ACTION ProcessInit_R1R2:
//*************************************************************************************************************
//
// build configuration for Instances and ProcessInterfaces
//
//*************************************************************************************************************
//*************************************************************************************************************
// - BufferInfeed     : single XtsStation which looks for input trigger from transfersystem, 
//                      transfersystem writes positions of XtsStations to be used at Infeed. 
//                      BufferInfeed is writing ItfProcessCollector[BufferInfeed.ProcessTarget].ActivateStation 
//                        for BufferInfeed target (Infeed / 12 XtsStations).
//                      BufferInfeed sends required amount of movers to WaitPos of XtsStations 
//                        of BufferInfeed target (Infeed / 12 XtsStations).
//-------------------------------------------------------------------------------------------------------------
// whoami
//
// process target (Infeed / 12 XtsStations)
//-------------------------------------------------------------------------------------------------------------
BufferInfeed.ProcessId                    := ProcessCollector[E_INSTANCE.BUFFER_INFEED].ProcessId;
BufferInfeed.ProcessTarget                := ProcessCollector[E_INSTANCE.INFEED].ProcessId;
BufferInfeed.CollectorInterface           := ItfProcessCollector;
BufferInfeed.ProcessLinkedLists           := ItfProcessList;
//-------------------------------------------------------------------------------------------------------------
// configure range of XtsStations for process
//
// see MAIN.StationParameterInit() for positions and dyn constraints
//-------------------------------------------------------------------------------------------------------------
ItfProcessCollector[BufferInfeed.ProcessId].StationFirst  := 53;
ItfProcessCollector[BufferInfeed.ProcessId].StationLast   := 53;

_nStnFrst                                 := ProcessCollector[BufferInfeed.ProcessId].StationFirst;
BufferInfeed.CheckPosition                := 15.0;

//-------------------------------------------------------------------------------------------------------------
//-------------------------------------------------------------------------------------------------------------
//*************************************************************************************************************
//*************************************************************************************************************
// - Infeed         : 12 XtsStations for transfersystem to unload
//                    Infeed is pulling in the movers according to list entry from BufferInfeed
//                    one stop only
//                    must be checked for all mover standstill in PosStop[1] of each XtsStation
//                    must be released by handshake from transfersystem (this is done by a TON for now)
//-------------------------------------------------------------------------------------------------------------
// whoami
//
// process target (BufferOutfeed / 1 XtsStation)
// TODO: 
//    configure infeed target for OUTFEED_CLAMP (12 XtsStations)
//    Infeed.ProcessTarget  := ProcessCollector[E_INSTANCE.OUTFEED_CLAMP].ProcessId;
//-------------------------------------------------------------------------------------------------------------
Infeed.ProcessId                          := ProcessCollector[E_INSTANCE.INFEED].ProcessId;
Infeed.ProcessTarget                      := ProcessCollector[E_INSTANCE.BUFFER_OUTFEED].ProcessId;
Infeed.CollectorInterface                 := ItfProcessCollector;
Infeed.ProcessLinkedLists                 := ItfProcessList;
//-------------------------------------------------------------------------------------------------------------
// configure range of XtsStations for process
//
// see MAIN.StationParameterInit() for positions and dyn constraints
//-------------------------------------------------------------------------------------------------------------
ItfProcessCollector[Infeed.ProcessId].StationFirst        :=  1;
ItfProcessCollector[Infeed.ProcessId].StationLast         := 12;
//-------------------------------------------------------------------------------------------------------------
//-------------------------------------------------------------------------------------------------------------
//*************************************************************************************************************
//*************************************************************************************************************
// - BufferOutfeed  : single XtsStation which distributes movers to specified range 
//                    Infeed sends all movers here 
//                    BufferOutfeed ensures that OutputR2 and OutputR1 have 12 movers each for every job
//                    BufferOutfeed checks if the Queue of this single XtsStation is empty or not
//-------------------------------------------------------------------------------------------------------------
// whoami
//
// process target (Outfeed (OutfeedR2 & OutfeedR1) / 24 XtsStations)
//
//  - optional process target (Outfeed 12 XtsStations)
//-------------------------------------------------------------------------------------------------------------
_nBufferOutfeedTarget[1] := E_INSTANCE.OUTFEED_ROBOT_R1;
_nBufferOutfeedTarget[2] := E_INSTANCE.OUTFEED_ROBOT_R2;

BufferOutfeed.ProcessId              := E_INSTANCE.BUFFER_OUTFEED;
BufferOutfeed.ProcessTarget          := _nBufferOutfeedTarget; 
BufferOutfeed.CollectorInterface     := ItfProcessCollector;
BufferOutfeed.ProcessLinkedLists     := ItfProcessList;
//-------------------------------------------------------------------------------------------------------------
// configure range of XtsStations for process
//
// see MAIN.StationParameterInit() for positions and dyn constraints
//-------------------------------------------------------------------------------------------------------------
ItfProcessCollector[BufferOutfeed.ProcessId].StationFirst  := 25;
ItfProcessCollector[BufferOutfeed.ProcessId].StationLast   := 25;

_nStnFrst                                 := ProcessCollector[BufferOutfeed.ProcessId].StationFirst;
BufferOutfeed.CheckPosition          := 2500.0;
//-------------------------------------------------------------------------------------------------------------
//-------------------------------------------------------------------------------------------------------------
//*************************************************************************************************************
//*************************************************************************************************************
// - Outfeed_R1  : 12 XtsStations for Robot 
//                    All XtsStations must be filled before robot can start 
//                    affter process all movers are sent to Sender process (high speed for the way back)
//                     
//                    
//-------------------------------------------------------------------------------------------------------------
// whoami
//
// process target (SenderFast / 1 XtsStation)
//-------------------------------------------------------------------------------------------------------------
Outfeed_R1.ProcessId                      := E_INSTANCE.OUTFEED_ROBOT_R1;
Outfeed_R1.ProcessTarget                  := ProcessCollector[E_INSTANCE.SENDER_FAST].ProcessId;
Outfeed_R1.CollectorInterface             := ItfProcessCollector;
Outfeed_R1.ProcessLinkedLists             := ItfProcessList;
//-------------------------------------------------------------------------------------------------------------
// configure range of XtsStations for process
//
// see MAIN.StationParameterInit() for positions and dyn constraints
//-------------------------------------------------------------------------------------------------------------
ItfProcessCollector[Outfeed_R1.ProcessId].StationFirst  := 26;
ItfProcessCollector[Outfeed_R1.ProcessId].StationLast   := 37;

_nStnFrst                                 := ProcessCollector[Outfeed_R1.ProcessId].StationFirst;
Outfeed_R1.CheckPosition                  := 6000.0;
//-------------------------------------------------------------------------------------------------------------
//-------------------------------------------------------------------------------------------------------------
//*************************************************************************************************************
//*************************************************************************************************************
// - Outfeed_R2  : 12 XtsStations for Robot 
//                    All XtsStations must be filled before robot can start 
//                    affter process all movers are sent to Sender process (high speed for the way back)
//                     
//                    
//-------------------------------------------------------------------------------------------------------------
// whoami
//
// process target (SenderFast / 1 XtsStation)
//-------------------------------------------------------------------------------------------------------------
Outfeed_R2.ProcessId                      := E_INSTANCE.OUTFEED_ROBOT_R2;
Outfeed_R2.ProcessTarget                  := ProcessCollector[E_INSTANCE.SENDER_FAST].ProcessId;
Outfeed_R2.CollectorInterface             := ItfProcessCollector;
Outfeed_R2.ProcessLinkedLists             := ItfProcessList;
//-------------------------------------------------------------------------------------------------------------
// configure range of XtsStations for process
//
// see MAIN.StationParameterInit() for positions and dyn constraints
//-------------------------------------------------------------------------------------------------------------
ItfProcessCollector[Outfeed_R2.ProcessId].StationFirst  := 38;
ItfProcessCollector[Outfeed_R2.ProcessId].StationLast   := 49;

_nStnFrst                                 := ProcessCollector[Outfeed_R2.ProcessId].StationFirst;
Outfeed_R2.CheckPosition                  := 6000.0;
//-------------------------------------------------------------------------------------------------------------
//-------------------------------------------------------------------------------------------------------------
//*************************************************************************************************************
//*************************************************************************************************************
// - SenderFast  : 1 XtsStation 
//                    movers are handled when entering position area 
//                    movers are accelerated to max speed
//                    movers do not stop here
//                    
//-------------------------------------------------------------------------------------------------------------
// whoami
//
// process target (SenderBufferInfeed / 1 XtsStation)
//-------------------------------------------------------------------------------------------------------------
SenderFast.ProcessId                      := E_INSTANCE.SENDER_FAST;
SenderFast.ProcessTarget                  := ProcessCollector[E_INSTANCE.SENDER_BUFFER_INFEED].ProcessId;
SenderFast.CollectorInterface             := ItfProcessCollector;
SenderFast.ProcessLinkedLists             := ItfProcessList;
//-------------------------------------------------------------------------------------------------------------
// configure range of XtsStations for process
//
// see MAIN.StationParameterInit() for positions and dyn constraints
//-------------------------------------------------------------------------------------------------------------
ItfProcessCollector[SenderFast.ProcessId].StationFirst  := 51;
ItfProcessCollector[SenderFast.ProcessId].StationLast   := 51;

_nStnFrst                                 := ProcessCollector[SenderFast.ProcessId].StationFirst;
SenderFast.CheckPosition                  := GVL_XTS.StationParameter[_nStnFrst].rPosWait - 500.0;
//-------------------------------------------------------------------------------------------------------------
//-------------------------------------------------------------------------------------------------------------
//*************************************************************************************************************
//*************************************************************************************************************
// - SenderBufferInfeed  : 1 XtsStation 
//                    movers are handled when entering position area 
//                    movers are sent to BufferInfeed, so that BufferInfeed has 12 mover ready
//                    movers do stop here, wait until there is room for movers
//                    
//-------------------------------------------------------------------------------------------------------------
// whoami
//
// process target (SenderBufferInfeed / 1 XtsStation)
//-------------------------------------------------------------------------------------------------------------
SenderBufferInfeed.ProcessId              := E_INSTANCE.SENDER_BUFFER_INFEED;
SenderBufferInfeed.ProcessTarget          := ProcessCollector[E_INSTANCE.BUFFER_INFEED].ProcessId;
SenderBufferInfeed.CollectorInterface     := ItfProcessCollector;
SenderBufferInfeed.ProcessLinkedLists     := ItfProcessList;
//-------------------------------------------------------------------------------------------------------------
// configure range of XtsStations for process
//
// see MAIN.StationParameterInit() for positions and dyn constraints
//-------------------------------------------------------------------------------------------------------------
ItfProcessCollector[SenderBufferInfeed.ProcessId].StationFirst  := 52;
ItfProcessCollector[SenderBufferInfeed.ProcessId].StationLast   := 52;

_nStnFrst                                 := ProcessCollector[SenderBufferInfeed.ProcessId].StationFirst;
SenderBufferInfeed.CheckPosition          := GVL_XTS.StationParameter[_nStnFrst].rPosWait - 1250.0;
//-------------------------------------------------------------------------------------------------------------
//-------------------------------------------------------------------------------------------------------------
//*************************************************************************************************************
END_ACTION

END_PROGRAM

// ---- MAIN.TcPOU
//---------------------------------------------------------------------------------------------------------------
//
//  HAUD 2024.03.18
//
//  - XTS_TRANSPORT_LAYER
//  - transport layer members:
//    - CaGroup
//      - access to Group functions
//
//    - Mover
//      - access to MC and CA motion functions
//
//    - Xpu (ProcessingUnit)
//      - access to TcCOM Objects in Environment
//
//    - Transport Control Unit
//      - coordinates members to get XTS in defined states
//
//    - Xts Stations
//      - handshakes with extern control for mover transport
//
//  - global datafields for mrmbers in GVL_XTS namespace
//  - global interface datafields for use in members
//  - structures are assigned by reference for every member
//
//---------------------------------------------------------------------------------------------------------------
// HAUD 2024 05 29
//
//    XTS_TRANSPORT_LAYER project
//    
//    MIT License
//    
//    Copyright (c) 2024 HAUD
//    
//    Permission is hereby granted, free of charge, to any person obtaining a copy
//    of this software and associated documentation files (the "Software"), to deal
//    in the Software without restriction, including without limitation the rights
//    to use, copy, modify, merge, publish, distribute, sublicense, and/or sell
//    copies of the Software, and to permit persons to whom the Software is
//    furnished to do so, subject to the following conditions:
//    
//    The above copyright notice and this permission notice shall be included in all
//    copies or substantial portions of the Software.
//    
//    THE SOFTWARE IS PROVIDED "AS IS", WITHOUT WARRANTY OF ANY KIND, EXPRESS OR
//    IMPLIED, INCLUDING BUT NOT LIMITED TO THE WARRANTIES OF MERCHANTABILITY,
//    FITNESS FOR A PARTICULAR PURPOSE AND NONINFRINGEMENT. IN NO EVENT SHALL THE
//    AUTHORS OR COPYRIGHT HOLDERS BE LIABLE FOR ANY CLAIM, DAMAGES OR OTHER
//    LIABILITY, WHETHER IN AN ACTION OF CONTRACT, TORT OR OTHERWISE, ARISING FROM,
//    OUT OF OR IN CONNECTION WITH THE SOFTWARE OR THE USE OR OTHER DEALINGS IN THE
//    SOFTWARE.
//---------------------------------------------------------------------------------------------------------------
PROGRAM MAIN
VAR
	bInit 				: BOOL;
  eInit         : E_PROGRESS;

  nStation,
	nMover,
  nMoverSelected,
  nStationSelected,
  nStationParameter   : UINT;

  sStationText        : STRING(30);

  eTransportState     : E_XTS_TRANSPORT_STATE;
  eTransportResult    : E_PROGRESS;

  eXpuState           : E_XPU_STATE;
  eXpuResult          : E_PROGRESS;
  eXpuCheck           : E_XPU_CHECK;

  eMoverState         : E_MOVER_STATE;
  eMoverResult        : E_PROGRESS;

  sCaGroupState,
  sTransportState,
  sTransportCheck,
  sTransportResult,
  sXpuState,
  sXpuResult,
  sXpuCheck,
  sXpuOpMode,
  sXpuMoverdetectionMode,
  sXpuMoverAssignement,
  sMoverState,
  sMoverResult,
  sStationState,
  sStationStateMask,
  sStationCtrlMask        : STRING;

  bStationEnable,
  bStationEnter,
  bStationStart,
  bStationDone,
  bStationOut,
  bStationGone            : BOOL;

  tStationSelectedQueue   : ARRAY[1..MAX_LIST_NODES] OF ST_STATION_MOVER_DATA;

  nStn                    : UINT;

  bWriteVariant           : BOOL;
  nParameterVariant       : UINT;
  rAcc                    : REAL := 30000.0;

  eMsgState                   : e_message_state;
  eMsgProgress                : E_PROGRESS;

  eMtrState                   : e_message_state;
  eMtrProgress                : E_PROGRESS;
END_VAR

//############################################################################
// Local time; used for timestamps
//############################################################################
GVL_MSG.fbLocalTime(
                    sLocalTime          => GVL_MSG.sLocalTime, 
                    dtLocalTime         => GVL_MSG.dtLocalTime);
//############################################################################
//############################################################################
// 	example for init sequence
//############################################################################	
IF NOT bInit
THEN
  CASE eInit
  OF
    E_PROGRESS.PROGRESS_INVALID,
    E_PROGRESS.PROGRESS_DONE:         // clear command interface
      eInit                                     := E_PROGRESS.PROGRESS_BUSY;
      GVL_XTS.XpuCtrl.Cmd                       := E_XPU_CTRL.XTS_CMD_NULL;
      GVL_MSG.TransportMessageCtrl.Cmd          := E_MESSAGE_CTRL.MSG_CTRL_NULL;
      GVL_MSG.MetricsMessageCtrl.Cmd            := E_MESSAGE_CTRL.MSG_CTRL_NULL;


      GVL_MSG.MessageLevelXpu                   := E_MessageType.eMessageVerbose; //GVL_MSG.MessageLevel;
      GVL_XTS.CaGroup.MessageLevel              := E_MessageType.eMessageVerbose; //GVL_MSG.MessageLevel;
      GVL_XTS.XtsTransport.MessageLevel         := E_MessageType.eMessageVerbose; //GVL_MSG.MessageLevel;

      FOR nStation := 1 TO MAX_STATION
      DO
        GVL_MSG.MessageLevelStations[nStation]  := E_MessageType.eMessageVerbose; //GVL_MSG.MessageLevel;
      END_FOR
      FOR nMover := 1 TO MAX_MOVER
      DO
        GVL_MSG.MessageLevelMovers[nMover]      := E_MessageType.eMessageVerbose; //GVL_MSG.MessageLevel;
      END_FOR


    E_PROGRESS.PROGRESS_BUSY:         // init Xpu, ProcessingUnit, MotorModules
      eInit                                     := E_PROGRESS.PROGRESS_PREPARE;
      GVL_XTS.XpuCtrl.Cmd                       := E_XPU_CTRL.XTS_CMD_INIT;
      GVL_MSG.TransportMessageCtrl.Cmd          := E_MESSAGE_CTRL.MSG_CTRL_INIT;
      GVL_MSG.MetricsMessageCtrl.Cmd            := E_MESSAGE_CTRL.MSG_CTRL_INIT;


    E_PROGRESS.PROGRESS_PREPARE:      // wait for init to be done
      IF (GVL_XTS.XpuState.State      = E_XPU_STATE.XTS_INIT + E_PROGRESS.PROGRESS_DONE)
      THEN
        eInit                                   := E_PROGRESS.PROGRESS_STARTUP;
        GVL_XTS.XpuCtrl.Cmd                     := E_XPU_CTRL.XTS_IDLE;
      END_IF

    E_PROGRESS.PROGRESS_STARTUP:      // check log file creation and assign mover interfaces
      IF (GVL_MSG.TransportMessageData.FileCreated) AND
         (GVL_MSG.MetricsMessageData.FileCreated)
      THEN
        eInit                                   := E_PROGRESS.PROGRESS_CHECK;
        GVL_MSG.TransportMessageCtrl.Cmd        := E_MESSAGE_CTRL.MSG_CTRL_IDLE;  // one local copy is made, no file is written
        GVL_MSG.MetricsMessageCtrl.Cmd          := E_MESSAGE_CTRL.MSG_CTRL_IDLE;  // one local copy is made, no file is written

        //---------------------------------------------------------------------------------------------------------------------
        // automated file write:
        //---------------------------------------------------------------------------------------------------------------------
        // GVL_MSG.TransportMessageCtrl.Cmd        := E_MESSAGE_CTRL.MSG_CTRL_NULL;  // MessageIndex and ErrorIndex are checked
        // GVL_MSG.MetricsMessageCtrl.Cmd          := E_MESSAGE_CTRL.MSG_CTRL_NULL;  // MessageIndex and ErrorIndex are checked
        //---------------------------------------------------------------------------------------------------------------------
        FOR nMover := 1 TO MAX_MOVER
        DO
          GVL_XTS.MoverItf[nMover]              := GVL_XTS.Mover[nMover];
        END_FOR
      END_IF

    E_PROGRESS.PROGRESS_CHECK:        // assign CaGroup interface
      eInit                                     := E_PROGRESS.PROGRESS_OCCUPIED;
      GVL_XTS.CaGroupItf                        := GVL_XTS.CaGroup;

    E_PROGRESS.PROGRESS_OCCUPIED:     // StartStation for XtsTransportCtrl.Cmd := E_XTS_TRANSPORT_CTRL.CMD_TRANSPORT_START;
      bWriteVariant                             := TRUE;
      eInit                                     := E_PROGRESS.PROGRESS_WORKING;

      // where to start?
      GVL_XTS.XtsTransport.StationStartIndex    := GVL_XTS.StationStartIndex;

      GVL_MSG.MessageLevelXpu                   := GVL_MSG.MessageLevel;
      GVL_XTS.CaGroup.MessageLevel              := GVL_MSG.MessageLevel;
      GVL_XTS.XtsTransport.MessageLevel         := GVL_MSG.MessageLevel;

      FOR nStation := 1 TO MAX_STATION
      DO
        GVL_MSG.MessageLevelStations[nStation]  := GVL_MSG.MessageLevel;
      END_FOR
      FOR nMover := 1 TO MAX_MOVER
      DO
        GVL_MSG.MessageLevelMovers[nMover]      := GVL_MSG.MessageLevel;
      END_FOR

    E_PROGRESS.PROGRESS_WORKING:
      // Start Position parameters
      GVL_XTS.StationStart.rPosWait             :=  20500.0; // this value may differ from the GVL_XTS.StationParameter[StartStationIndex], IF it differs, you MUST have room for positive movement to GVL_XTS.StationParameter[StartStationIndex].rWaitPos
      GVL_XTS.StationStart.rGap                 :=     85.0; // may differ, or just copy from GVL_XTS.StationParameter[StartStationIndex]
      GVL_XTS.StationStart.rVelo                :=   1250.0; // may differ, or just copy from GVL_XTS.StationParameter[StartStationIndex]
      GVL_XTS.StationStart.rAccDec              :=  15000.0; // may differ, or just copy from GVL_XTS.StationParameter[StartStationIndex]
      GVL_XTS.StationStart.rJerk                := 400000.0; // may differ, or just copy from GVL_XTS.StationParameter[StartStationIndex], the movements are more robust if you keep this value in a narrow range, since jumps lead to adjusting movements within the CA Group

      IF (GVL_XTS.XtsTransport.StationStartIndex > 0) AND
         (GVL_XTS.XtsTransport.StationStartIndex < MAX_STATION+1)
      THEN
        GVL_XTS.StationStart.nConfiguredStopCount := GVL_XTS.StationParameter[GVL_XTS.XtsTransport.StationStartIndex].nConfiguredStopCount;
      END_IF

      bInit                                     := TRUE;
      eInit                                     := E_PROGRESS.PROGRESS_DONE;
  END_CASE
END_IF
//############################################################################
//############################################################################
// 	XTS Transport Unit
//############################################################################
//  - main control function block for transport layer
//  - requires access to member controls
//    - Xpu
//    - CaGroup
//    - Mover
//    - Station Control
//    - Station LinkedList Interface
//############################################################################
//
// cyclic call
GVL_XTS.XtsTransport();

// main control
GVL_XTS.XtsTransport.Ctrl               REF= GVL_XTS.XtsTransportCtrl;   // main control
GVL_XTS.XtsTransport.State              REF= GVL_XTS.XtsTransportState;  // main state
                                        
// member controls                      
GVL_XTS.XtsTransport.XpuCtrl            REF= GVL_XTS.XpuCtrl;
GVL_XTS.XtsTransport.XpuState           REF= GVL_XTS.XpuState;
GVL_XTS.XtsTransport.XpuInfo            REF= GVL_XTS.XpuInfo;
                                        
GVL_XTS.XtsTransport.GroupItf           :=   GVL_XTS.CaGroupItf;
GVL_XTS.XtsTransport.GroupInfo          REF= GVL_XTS.CaGroupInfo;
                                        
GVL_XTS.XtsTransport.MoverItf           REF= GVL_XTS.MoverItf;
GVL_XTS.XtsTransport.MoverInfo          REF= GVL_XTS.MoverInfo;
GVL_XTS.XtsTransport.MoverLastPosition  REF= GVL_XTS.LastPosition;
GVL_XTS.XtsTransport.MoverLastGap       REF= GVL_XTS.LastGap;
                                        
GVL_XTS.XtsTransport.StationStart       REF= GVL_XTS.StationStart;      // start position for E_XTS_TRANSPORT_CTRL.CMD_TRANSPORT_START
GVL_XTS.XtsTransport.StationCtrlItf     REF= GVL_XTS.StationCtrlItf;    // station interfaces are required for accessing station methods
GVL_XTS.XtsTransport.StationListsItf    REF= GVL_XTS.StationListItf;    // list interface is required for access to linked list methods
GVL_XTS.XtsTransport.StationControl     REF= GVL_XTS.StationCtrl;
GVL_XTS.XtsTransport.StationState       REF= GVL_XTS.StationState;
//############################################################################



//############################################################################
// 	XTS Stations
//############################################################################	
FOR nStation := 1 TO MAX_STATION
DO
  GVL_XTS.Station[nStation].StationId   := nStation;
  GVL_XTS.Station[nStation].MessageLevel:= GVL_MSG.MessageLevelStations[nStation];

  GVL_XTS.StationListItf[nStation]      := GVL_XTS.StationList[nStation];   // interfaces for list methods
  GVL_XTS.StationCtrlItf[nStation]      := GVL_XTS.Station[nStation];       // interfaces for station methods

  GVL_XTS.Station[nStation].Ctrl        REF= GVL_XTS.StationCtrl;           // station ctrl from extern
  GVL_XTS.Station[nStation].State       REF= GVL_XTS.StationState;          // station state to extern

  GVL_XTS.Station[nStation].ItfStations REF= GVL_XTS.StationListItf;        // give every station all list interfaces for writing mover tickets
  GVL_XTS.Station[nStation].ItfMover    REF= GVL_XTS.MoverItf;              // give every station all mover interfaces for movement in / out of station
  GVL_XTS.Station[nStation].Mover       REF= GVL_XTS.AxisRefMover;          // AXIS_REF to read infos from
  GVL_XTS.Station[nStation].MoverOffset REF= GVL_XTS.PositionOffset;        // static offsets for all stations, all movers, all stop positions


  GVL_XTS.Station[nStation].StationParameter  REF= GVL_XTS.StationParameter;// give every station all station parameters for sending to WaitPos of target station

  // cyclic call
  GVL_XTS.Station[nStation].Cycle();                                        // cycle for handshaking with extern

  // Queue data for each station
  GVL_XTS.StationQueue[nStation]        := GVL_XTS.StationListItf[nStation].Data;
END_FOR
//############################################################################



//############################################################################
// 	XPU environment
//############################################################################	
GVL_XTS.Xpu.XpuInstance                 :=   1;
GVL_XTS.Xpu.MessageLevel                :=   GVL_MSG.MessageLevelXpu;

GVL_XTS.Xpu.Ctrl                        REF= GVL_XTS.XpuCtrl;
GVL_XTS.Xpu.State                       REF= GVL_XTS.XpuState;
GVL_XTS.Xpu.XpuModuleInfoData           REF= GVL_XTS.XpuModules;

GVL_XTS.Xpu.CaGroupOID                  :=   GVL_XTS.CaGroup.GroupInfo.CaGroupOID;

// cyclic call
GVL_XTS.Xpu();
GVL_XTS.XpuInfo                         :=   GVL_XTS.Xpu.XpuInfo;
//############################################################################


//############################################################################	
// 	CA-Group Class
//############################################################################	
// assignment
GVL_XTS.CaGroup.AxisRef                 REF= GVL_XTS.AxisRefMover;
// Interface to Mover methods
GVL_XTS.CaGroup.MoverItf                REF= GVL_XTS.MoverItf; 

GVL_XTS.CaGroup.GroupRef                REF= GVL_XTS.CaGroupRef;

// cyclic call
GVL_XTS.CaGroup.InfoCycle(TRUE); // read group status

// InfoData from group
GVL_XTS.CaGroupInfo                     :=   GVL_XTS.CaGroup.GroupInfo;

// Interface of CaGroup
GVL_XTS.CaGroupItf                      :=   GVL_XTS.CaGroup;
//############################################################################


//############################################################################
// Mover Class	
//############################################################################	
FOR nMover := 1 TO MAX_MOVER
DO
  GVL_XTS.Mover[nMover].MoverId         :=   nMover;
  GVL_XTS.Mover[nMover].RailLength      :=   GVL_XTS.Xpu.RailLength;  // mover needs RailLength, in order to calc absolute position from modulo input
  GVL_XTS.Mover[nMover].MessageLevel    :=   GVL_MSG.MessageLevelMovers[nMover];

  GVL_XTS.Mover[nMover].Ctrl            REF= GVL_XTS.MoverCtrl;       // mover control from extern
  GVL_XTS.Mover[nMover].State           REF= GVL_XTS.MoverState;      // mover state to extern

  GVL_XTS.Mover[nMover].MoveData        REF= GVL_XTS.MoveData;        // dyn constraints for extern to write
  GVL_XTS.Mover[nMover].GearData        REF= GVL_XTS.GearData;        // GearIn/GearInPosCa data fro extern to write

  // assignment	
  GVL_XTS.Mover[nMover].Mover           REF= GVL_XTS.AxisRefMover[nMover];  // axis reference to Mover function block
  GVL_XTS.Mover[nMover].LastGap         REF= GVL_XTS.LastGap[nMover];       // reference to last used gap value datafield
  GVL_XTS.Mover[nMover].LastPosition    REF= GVL_XTS.LastPosition[nMover];  // reference to last position datafield

  GVL_XTS.Mover[nMover].MoverInfo		    REF= GVL_XTS.MoverInfo[nMover];     // refernence to mover info data (ActPos, SetPos, ...)

  GVL_XTS.MoverItf[nMover]              :=   GVL_XTS.Mover[nMover];

  // cyclic call
  GVL_XTS.Mover[nMover].Cycle();  // call AXIS_REF()
  GVL_XTS.Mover[nMover]();        // call Ctrl/State
END_FOR
//############################################################################
//############################################################################
// /logging
//############################################################################
GVL_MSG.TransportMessageData.Ctrl             REF= GVL_MSG.TransportMessageCtrl;
GVL_MSG.TransportMessageData.State            REF= GVL_MSG.TransportMessageState;

GVL_MSG.TransportMessageData.MessageIndex     REF= GVL_MSG.MessageTransportIndex;
GVL_MSG.TransportMessageData.ErrorIndex       REF= GVL_MSG.MessageTransportError;

GVL_MSG.TransportMessageData.DirRoot          :=   ADR(GVL_MSG.LOG_DIR);
GVL_MSG.TransportMessageData.FileRoot         :=   ADR(GVL_MSG.LOG_FILE);

GVL_MSG.TransportMessageData.MsgList          :=   ADR(GVL_MSG.TransportMessages);
GVL_MSG.TransportMessageData.LocalTime        :=   ADR(GVL_MSG.dtLocalTime);

GVL_MSG.TransportMessageData();               

eMsgState                                     := f_GetState   (GVL_MSG.TransportMessageState.State);
eMsgProgress                                  := f_GetProgress(GVL_MSG.TransportMessageState.State);

CASE eMsgState
OF
  E_MESSAGE_STATE.MSG_STATE_NULL:
    CASE eMsgProgress
    OF
      E_PROGRESS.PROGRESS_INVALID,
      E_PROGRESS.PROGRESS_DONE:
        IF (GVL_MSG.MessageTransportIndex > GVL_MSG.MAX_MESSAGE/100) OR
           (GVL_MSG.MessageTransportError > 0)
        THEN
          GVL_MSG.TransportMessageCtrl.Cmd    := E_MESSAGE_CTRL.MSG_CTRL_WRITE;
        END_IF
    END_CASE

  E_MESSAGE_STATE.MSG_STATE_WRITE:
    CASE eMsgProgress
    OF
      E_PROGRESS.PROGRESS_ERROR,
      E_PROGRESS.PROGRESS_DONE:
        GVL_MSG.TransportMessageCtrl.Cmd      := E_MESSAGE_CTRL.MSG_CTRL_NULL;
    END_CASE

ELSE
    CASE eMsgProgress
    OF
      E_PROGRESS.PROGRESS_DONE:
        GVL_MSG.TransportMessageCtrl.Cmd      := E_MESSAGE_CTRL.MSG_CTRL_NULL;
    END_CASE
END_CASE
//############################################################################
// logging/
//############################################################################
//############################################################################
//############################################################################
// /Transport Metrics
//############################################################################
GVL_MSG.MetricsMessageData.Ctrl               REF= GVL_MSG.MetricsMessageCtrl;
GVL_MSG.MetricsMessageData.State              REF= GVL_MSG.MetricsMessageState;

GVL_MSG.MetricsMessageData.MessageIndex       REF= GVL_MSG.MessageMetricsIndex;
GVL_MSG.MetricsMessageData.ErrorIndex         REF= GVL_MSG.MessageMetricsError;

GVL_MSG.MetricsMessageData.DirRoot            :=   ADR(GVL_MSG.LOG_DIR);
GVL_MSG.MetricsMessageData.FileRoot           :=   ADR(GVL_MSG.LOG_FILE_METRIC);

GVL_MSG.MetricsMessageData.MsgList            :=   ADR(GVL_MSG.MetricsMessages);
GVL_MSG.MetricsMessageData.LocalTime          :=   ADR(GVL_MSG.dtLocalTime);

GVL_MSG.MetricsMessageData();

eMtrState                                     := f_GetState   (GVL_MSG.MetricsMessageState.State);
eMtrProgress                                  := f_GetProgress(GVL_MSG.MetricsMessageState.State);

CASE eMtrState
OF
  E_MESSAGE_STATE.MSG_STATE_NULL:
    CASE eMtrProgress
    OF
      E_PROGRESS.PROGRESS_INVALID:
        IF (GVL_MSG.MessageMetricsIndex > 10) OR
           (GVL_MSG.MessageMetricsError > 0)
        THEN
          GVL_MSG.MetricsMessageCtrl.Cmd      := E_MESSAGE_CTRL.MSG_CTRL_WRITE;
        END_IF
    END_CASE

  E_MESSAGE_STATE.MSG_STATE_WRITE:
    CASE eMtrProgress
    OF
      E_PROGRESS.PROGRESS_ERROR,
      E_PROGRESS.PROGRESS_DONE:
        GVL_MSG.MetricsMessageCtrl.Cmd        := E_MESSAGE_CTRL.MSG_CTRL_NULL;
    END_CASE
ELSE
    CASE eMtrProgress
    OF
      E_PROGRESS.PROGRESS_DONE:
        GVL_MSG.MetricsMessageCtrl.Cmd        := E_MESSAGE_CTRL.MSG_CTRL_NULL;
    END_CASE
END_CASE
//############################################################################
// Transport Metrics/
//############################################################################
//############################################################################
//############################################################################
// Visualization data	
//############################################################################	
// get enumerations from XPU for visu:
eTransportState                         := f_GetState   (GVL_XTS.XtsTransportState.State);
eTransportResult                        := f_GetProgress(GVL_XTS.XtsTransportState.State);

eXpuState                               := f_GetState   (GVL_XTS.XpuState.State);
eXpuResult                              := f_GetProgress(GVL_XTS.XpuState.State);

eXpuCheck                               := GVL_XTS.XpuState.Check;

// display xpu state and result in visu
// get strings and info
sCaGroupState                           := TO_STRING(GVL_XTS.CaGroupInfo.CaGroupState);

sTransportState                         := TO_STRING(eTransportState);
sTransportCheck                         := TO_STRING(GVL_XTS.XtsTransportState.Check);
sTransportResult                        := TO_STRING(eTransportResult);

sXpuState                               := TO_STRING(eXpuState);
sXpuResult                              := TO_STRING(eXpuResult);
sXpuCheck                               := TO_STRING(eXpuCheck);

sXpuOpMode                              := GVL_XTS.Xpu.OpModeToString();
sXpuMoverdetectionMode                  := GVL_XTS.Xpu.IdDetectionModeToString();
sXpuMoverAssignement                    := GVL_XTS.Xpu.MoverPositionAssignementToString();

nMoverSelected                          := SEL((nMoverSelected<1), nMoverSelected, 1);
nMoverSelected                          := SEL((nMoverSelected>MAX_MOVER), nMoverSelected, MAX_MOVER);

nStationSelected                        := SEL((nStationSelected<1), nStationSelected, 1);
nStationSelected                        := SEL((nStationSelected>MAX_STATION), nStationSelected, MAX_STATION);

bStationEnable                          := SEL((GVL_XTS.StationCtrl[nStationSelected].eCmd = E_STATION_CTRL.STATION_ENABLE),        FALSE, TRUE);
bStationEnter                           := SEL((GVL_XTS.StationCtrl[nStationSelected].eCmd = E_STATION_CTRL.STATION_MOVER_ENTER),   FALSE, TRUE);
bStationStart                           := SEL((GVL_XTS.StationCtrl[nStationSelected].eCmd = E_STATION_CTRL.STATION_PROCESS_START), FALSE, TRUE);
bStationDone                            := SEL((GVL_XTS.StationCtrl[nStationSelected].eCmd = E_STATION_CTRL.STATION_PROCESS_DONE),  FALSE, TRUE);
bStationOut                             := SEL((GVL_XTS.StationCtrl[nStationSelected].eCmd = E_STATION_CTRL.STATION_MOVER_OUT),     FALSE, TRUE);
bStationGone                            := SEL((GVL_XTS.StationCtrl[nStationSelected].eCmd = E_STATION_CTRL.STATION_MOVER_GONE),    FALSE, TRUE);

eMoverState                             := f_GetState   (GVL_XTS.MoverState[nMoverSelected].State);
eMoverResult                            := f_GetProgress(GVL_XTS.MoverState[nMoverSelected].State);

sMoverState                             := TO_STRING(eMoverState);
sMoverResult                            := TO_STRING(eMoverResult);

sStationState                           := TO_STRING(GVL_XTS.StationState[nStationSelected].eState);
sStationStateMask                       := Tc2_Utilities.BYTE_TO_BINSTR(GVL_XTS.StationState[nStationSelected].nMask, 8);
sStationCtrlMask                        := Tc2_Utilities.BYTE_TO_BINSTR(GVL_XTS.StationCtrl[nStationSelected].nMask, 8);

tStationSelectedQueue                   := GVL_XTS.StationQueue[nStationSelected];

IF bWriteVariant
THEN
  bWriteVariant                         := FALSE;

  CASE nParameterVariant
  OF
    1:
      J_100000_V3000();     // J 100_000 V3000
    2:
      J_100000_V3500();     // J 100_000 V3500
    3:
      J_100000_V4000();     // J 100_000 V4000
    4:
      J_200000_V3000();     // J 200_000 V3000
    5:
      StationParameterInit_4();   // J 400_000
    6:
      StationParameterInit_5();   // J 100_000 PosStop INFEED == 0.0
  ELSE
      StationParameterInit_5();   // J 100_000 PosStop INFEED == 0.0
  END_CASE
END_IF
//############################################################################
//############################################################################

ACTION J_100000_V3000:
//-----------------------------------------------------------------------------
//
//  HAUD 2024.06.12
//
// 
//  - hard coded station parameter
//-----------------------------------------------------------------------------
//-----------------------------------------------------------------------------

FOR nStationParameter := 1 TO MAX_STATION
DO
  GVL_XTS.StationParameter[nStationParameter].rVelo               :=   3000.0;
  GVL_XTS.StationParameter[nStationParameter].rAccDec             := rAcc;
  GVL_XTS.StationParameter[nStationParameter].rJerk               := 100000.0;
END_FOR 

//-----------------------------------------------------------------------------------------------------------------------------------------
//  INFEED
    sStationText  := TO_STRING(E_INSTANCE.INFEED);//'INFEED';
//-----------------------------------------------------------------------------------------------------------------------------------------
nStationParameter := 1;
GVL_XTS.StationParameter[nStationParameter].sText                 := sStationText;
GVL_XTS.StationParameter[nStationParameter].rPosWait              :=    1250.0;  // absolute modulo position

GVL_XTS.StationParameter[nStationParameter].nConfiguredStopCount  :=      1;   // how many stops the mover has to make in this station
GVL_XTS.StationParameter[nStationParameter].rPosStop[1]           :=      0.0 + 176.0; // relative to rPosWait

GVL_XTS.StationParameter[nStationParameter].rReleaseDistance      :=    300.0; // relative to Mover.ActPos
GVL_XTS.StationParameter[nStationParameter].rGap                  :=     76.0;

//-----------------------------------------------------------------------------------------------------------------------------------------
nStationParameter := 2;
GVL_XTS.StationParameter[nStationParameter].sText                 := sStationText;
GVL_XTS.StationParameter[nStationParameter].rPosWait              :=    1250.0; // absolute modulo position

GVL_XTS.StationParameter[nStationParameter].nConfiguredStopCount  :=      1;   // how many stops the mover has to make in this station
GVL_XTS.StationParameter[nStationParameter].rPosStop[1]           :=     76.0 + 176.0; // relative to rPosWait

GVL_XTS.StationParameter[nStationParameter].rReleaseDistance      :=    275.0; // relative to Mover.ActPos
GVL_XTS.StationParameter[nStationParameter].rGap                  :=     76.0;

//-----------------------------------------------------------------------------------------------------------------------------------------
nStationParameter := 3;
GVL_XTS.StationParameter[nStationParameter].sText                 := sStationText;
GVL_XTS.StationParameter[nStationParameter].rPosWait              :=    1250.0; // absolute modulo position

GVL_XTS.StationParameter[nStationParameter].nConfiguredStopCount  :=      1;   // how many stops the mover has to make in this station
GVL_XTS.StationParameter[nStationParameter].rPosStop[1]           :=    152.0 + 176.0; // relative to rPosWait

GVL_XTS.StationParameter[nStationParameter].rReleaseDistance      :=    250.0; // relative to Mover.ActPos
GVL_XTS.StationParameter[nStationParameter].rGap                  :=     76.0;

//-----------------------------------------------------------------------------------------------------------------------------------------
nStationParameter := 4;
GVL_XTS.StationParameter[nStationParameter].sText                 := sStationText;
GVL_XTS.StationParameter[nStationParameter].rPosWait              :=   1250.0;  // absolute modulo position

GVL_XTS.StationParameter[nStationParameter].nConfiguredStopCount  :=      1;   // how many stops the mover has to make in this station
GVL_XTS.StationParameter[nStationParameter].rPosStop[1]           :=    228.0 + 176.0; // relative to rPosWait

GVL_XTS.StationParameter[nStationParameter].rReleaseDistance      :=    225.0; // relative to Mover.ActPos
GVL_XTS.StationParameter[nStationParameter].rGap                  :=     76.0;

//-----------------------------------------------------------------------------------------------------------------------------------------
nStationParameter := 5;
GVL_XTS.StationParameter[nStationParameter].sText                 := sStationText;
GVL_XTS.StationParameter[nStationParameter].rPosWait              :=   1250.0;  // absolute modulo position

GVL_XTS.StationParameter[nStationParameter].nConfiguredStopCount  :=      1;   // how many stops the mover has to make in this station
GVL_XTS.StationParameter[nStationParameter].rPosStop[1]           :=    304.0 + 176.0; // relative to rPosWait

GVL_XTS.StationParameter[nStationParameter].rReleaseDistance      :=    200.0; // relative to Mover.ActPos
GVL_XTS.StationParameter[nStationParameter].rGap                  :=     76.0;

//-----------------------------------------------------------------------------------------------------------------------------------------
nStationParameter := 6;
GVL_XTS.StationParameter[nStationParameter].sText                 := sStationText;
GVL_XTS.StationParameter[nStationParameter].rPosWait              :=   1250.0;  // absolute modulo position

GVL_XTS.StationParameter[nStationParameter].nConfiguredStopCount  :=      1;   // how many stops the mover has to make in this station
GVL_XTS.StationParameter[nStationParameter].rPosStop[1]           :=    380.0 + 176.0; // relative to rPosWait

GVL_XTS.StationParameter[nStationParameter].rReleaseDistance      :=    175.0; // relative to Mover.ActPos
GVL_XTS.StationParameter[nStationParameter].rGap                  :=     76.0;

//-----------------------------------------------------------------------------------------------------------------------------------------
nStationParameter := 7;
GVL_XTS.StationParameter[nStationParameter].sText                 := sStationText;
GVL_XTS.StationParameter[nStationParameter].rPosWait              :=   1250.0;  // absolute modulo position

GVL_XTS.StationParameter[nStationParameter].nConfiguredStopCount  :=      1;   // how many stops the mover has to make in this station
GVL_XTS.StationParameter[nStationParameter].rPosStop[1]           :=    456.0 + 176.0; // relative to rPosWait

GVL_XTS.StationParameter[nStationParameter].rReleaseDistance      :=    150.0; // relative to Mover.ActPos
GVL_XTS.StationParameter[nStationParameter].rGap                  :=     76.0;

//-----------------------------------------------------------------------------------------------------------------------------------------
nStationParameter := 8;
GVL_XTS.StationParameter[nStationParameter].sText                 := sStationText;
GVL_XTS.StationParameter[nStationParameter].rPosWait              :=   1250.0;  // absolute modulo position

GVL_XTS.StationParameter[nStationParameter].nConfiguredStopCount  :=      1;   // how many stops the mover has to make in this station
GVL_XTS.StationParameter[nStationParameter].rPosStop[1]           :=    532.0 + 176.0; // relative to rPosWait

GVL_XTS.StationParameter[nStationParameter].rReleaseDistance      :=    125.0; // relative to Mover.ActPos
GVL_XTS.StationParameter[nStationParameter].rGap                  :=     76.0;

//-----------------------------------------------------------------------------------------------------------------------------------------
nStationParameter := 9;
GVL_XTS.StationParameter[nStationParameter].sText                 := sStationText;
GVL_XTS.StationParameter[nStationParameter].rPosWait              :=   1250.0;  // absolute modulo position

GVL_XTS.StationParameter[nStationParameter].nConfiguredStopCount  :=      1;   // how many stops the mover has to make in this station
GVL_XTS.StationParameter[nStationParameter].rPosStop[1]           :=    608.0 + 176.0; // relative to rPosWait

GVL_XTS.StationParameter[nStationParameter].rReleaseDistance      :=    100.0; // relative to Mover.ActPos
GVL_XTS.StationParameter[nStationParameter].rGap                  :=     76.0;

//-----------------------------------------------------------------------------------------------------------------------------------------
nStationParameter := 10;
GVL_XTS.StationParameter[nStationParameter].sText                 := sStationText;
GVL_XTS.StationParameter[nStationParameter].rPosWait              :=   1250.0;  // absolute modulo position

GVL_XTS.StationParameter[nStationParameter].nConfiguredStopCount  :=      1;   // how many stops the mover has to make in this station
GVL_XTS.StationParameter[nStationParameter].rPosStop[1]           :=    684.0 + 176.0; // relative to rPosWait

GVL_XTS.StationParameter[nStationParameter].rReleaseDistance      :=     75.0; // relative to Mover.ActPos
GVL_XTS.StationParameter[nStationParameter].rGap                  :=     76.0;

//-----------------------------------------------------------------------------------------------------------------------------------------
nStationParameter := 11;
GVL_XTS.StationParameter[nStationParameter].sText                 := sStationText;
GVL_XTS.StationParameter[nStationParameter].rPosWait              :=   1250.0;  // absolute modulo position

GVL_XTS.StationParameter[nStationParameter].nConfiguredStopCount  :=      1;   // how many stops the mover has to make in this station
GVL_XTS.StationParameter[nStationParameter].rPosStop[1]           :=    760.0 + 176.0; // relative to rPosWait

GVL_XTS.StationParameter[nStationParameter].rReleaseDistance      :=     50.0; // relative to Mover.ActPos
GVL_XTS.StationParameter[nStationParameter].rGap                  :=     76.0;

//-----------------------------------------------------------------------------------------------------------------------------------------
nStationParameter := 12;
GVL_XTS.StationParameter[nStationParameter].sText                 := sStationText;
GVL_XTS.StationParameter[nStationParameter].rPosWait              :=   1250.0;  // absolute modulo position

GVL_XTS.StationParameter[nStationParameter].nConfiguredStopCount  :=      1;   // how many stops the mover has to make in this station
GVL_XTS.StationParameter[nStationParameter].rPosStop[1]           :=    836.0 + 176.0; // relative to rPosWait

GVL_XTS.StationParameter[nStationParameter].rReleaseDistance      :=     10.0; // relative to Mover.ActPos
GVL_XTS.StationParameter[nStationParameter].rGap                  :=     76.0;

//-----------------------------------------------------------------------------------------------------------------------------------------
//-----------------------------------------------------------------------------------------------------------------------------------------
//  OUTFEED_CLAMP (not in use in this example)
    sStationText  := 'OUTFEED_CLAMP';
//-----------------------------------------------------------------------------------------------------------------------------------------
nStationParameter := 13;
GVL_XTS.StationParameter[nStationParameter].sText                 := sStationText;
GVL_XTS.StationParameter[nStationParameter].rPosWait              :=   3582.0;  // absolute modulo position

GVL_XTS.StationParameter[nStationParameter].nConfiguredStopCount  :=      1;   // how many stops the mover has to make in this station
GVL_XTS.StationParameter[nStationParameter].rPosStop[1]           :=      0.0 + 161.0; // relative to rPosWait

GVL_XTS.StationParameter[nStationParameter].rReleaseDistance      :=    120.0; // relative to Mover.ActPos
GVL_XTS.StationParameter[nStationParameter].rGap                  :=     76.0;

//-----------------------------------------------------------------------------------------------------------------------------------------
nStationParameter := 14;
GVL_XTS.StationParameter[nStationParameter].sText                 := sStationText;
GVL_XTS.StationParameter[nStationParameter].rPosWait              :=   3582.0;  // absolute modulo position

GVL_XTS.StationParameter[nStationParameter].nConfiguredStopCount  :=      1;   // how many stops the mover has to make in this station
GVL_XTS.StationParameter[nStationParameter].rPosStop[1]           :=     76.0 + 161.0; // relative to rPosWait

GVL_XTS.StationParameter[nStationParameter].rReleaseDistance      :=    110.0; // relative to Mover.ActPos
GVL_XTS.StationParameter[nStationParameter].rGap                  :=     76.0;

//-----------------------------------------------------------------------------------------------------------------------------------------
nStationParameter := 15;
GVL_XTS.StationParameter[nStationParameter].sText                 := sStationText;
GVL_XTS.StationParameter[nStationParameter].rPosWait              :=   3582.0;  // absolute modulo position

GVL_XTS.StationParameter[nStationParameter].nConfiguredStopCount  :=      1;   // how many stops the mover has to make in this station
GVL_XTS.StationParameter[nStationParameter].rPosStop[1]           :=    152.0 + 161.0; // relative to rPosWait

GVL_XTS.StationParameter[nStationParameter].rReleaseDistance      :=    100.0; // relative to Mover.ActPos
GVL_XTS.StationParameter[nStationParameter].rGap                  :=     76.0;

//-----------------------------------------------------------------------------------------------------------------------------------------
nStationParameter := 16;
GVL_XTS.StationParameter[nStationParameter].sText                 := sStationText;
GVL_XTS.StationParameter[nStationParameter].rPosWait              :=   3582.0;  // absolute modulo position

GVL_XTS.StationParameter[nStationParameter].nConfiguredStopCount  :=      1;   // how many stops the mover has to make in this station
GVL_XTS.StationParameter[nStationParameter].rPosStop[1]           :=    228.0 + 161.0; // relative to rPosWait

GVL_XTS.StationParameter[nStationParameter].rReleaseDistance      :=     90.0; // relative to Mover.ActPos
GVL_XTS.StationParameter[nStationParameter].rGap                  :=     76.0;

//-----------------------------------------------------------------------------------------------------------------------------------------
nStationParameter := 17;
GVL_XTS.StationParameter[nStationParameter].sText                 := sStationText;
GVL_XTS.StationParameter[nStationParameter].rPosWait              :=   3582.0;  // absolute modulo position

GVL_XTS.StationParameter[nStationParameter].nConfiguredStopCount  :=      1;   // how many stops the mover has to make in this station
GVL_XTS.StationParameter[nStationParameter].rPosStop[1]           :=    304.0 + 161.0; // relative to rPosWait

GVL_XTS.StationParameter[nStationParameter].rReleaseDistance      :=     80.0; // relative to Mover.ActPos
GVL_XTS.StationParameter[nStationParameter].rGap                  :=     76.0;

//-----------------------------------------------------------------------------------------------------------------------------------------
nStationParameter := 18;
GVL_XTS.StationParameter[nStationParameter].sText                 := sStationText;
GVL_XTS.StationParameter[nStationParameter].rPosWait              :=   3582.0;  // absolute modulo position

GVL_XTS.StationParameter[nStationParameter].nConfiguredStopCount  :=      1;   // how many stops the mover has to make in this station
GVL_XTS.StationParameter[nStationParameter].rPosStop[1]           :=    380.0 + 161.0; // relative to rPosWait

GVL_XTS.StationParameter[nStationParameter].rReleaseDistance      :=     70.0; // relative to Mover.ActPos
GVL_XTS.StationParameter[nStationParameter].rGap                  :=     76.0;

//-----------------------------------------------------------------------------------------------------------------------------------------
nStationParameter := 19;
GVL_XTS.StationParameter[nStationParameter].sText                 := sStationText;
GVL_XTS.StationParameter[nStationParameter].rPosWait              :=   3582.0;  // absolute modulo position

GVL_XTS.StationParameter[nStationParameter].nConfiguredStopCount  :=      1;   // how many stops the mover has to make in this station
GVL_XTS.StationParameter[nStationParameter].rPosStop[1]           :=    456.0 + 161.0; // relative to rPosWait

GVL_XTS.StationParameter[nStationParameter].rReleaseDistance      :=     60.0; // relative to Mover.ActPos
GVL_XTS.StationParameter[nStationParameter].rGap                  :=     76.0;

//-----------------------------------------------------------------------------------------------------------------------------------------
nStationParameter := 20;
GVL_XTS.StationParameter[nStationParameter].sText                 := sStationText;
GVL_XTS.StationParameter[nStationParameter].rPosWait              :=   3582.0;  // absolute modulo position

GVL_XTS.StationParameter[nStationParameter].nConfiguredStopCount  :=      1;   // how many stops the mover has to make in this station
GVL_XTS.StationParameter[nStationParameter].rPosStop[1]           :=    532.0 + 161.0; // relative to rPosWait

GVL_XTS.StationParameter[nStationParameter].rReleaseDistance      :=     50.0; // relative to Mover.ActPos
GVL_XTS.StationParameter[nStationParameter].rGap                  :=     76.0;

//-----------------------------------------------------------------------------------------------------------------------------------------
nStationParameter := 21;
GVL_XTS.StationParameter[nStationParameter].sText                 := sStationText;
GVL_XTS.StationParameter[nStationParameter].rPosWait              :=   3582.0;  // absolute modulo position

GVL_XTS.StationParameter[nStationParameter].nConfiguredStopCount  :=      1;   // how many stops the mover has to make in this station
GVL_XTS.StationParameter[nStationParameter].rPosStop[1]           :=    608.0 + 161.0; // relative to rPosWait

GVL_XTS.StationParameter[nStationParameter].rReleaseDistance      :=     40.0; // relative to Mover.ActPos
GVL_XTS.StationParameter[nStationParameter].rGap                  :=     76.0;

//-----------------------------------------------------------------------------------------------------------------------------------------
nStationParameter := 22;
GVL_XTS.StationParameter[nStationParameter].sText                 := sStationText;
GVL_XTS.StationParameter[nStationParameter].rPosWait              :=   3582.0;  // absolute modulo position

GVL_XTS.StationParameter[nStationParameter].nConfiguredStopCount  :=      1;   // how many stops the mover has to make in this station
GVL_XTS.StationParameter[nStationParameter].rPosStop[1]           :=    684.0 + 161.0; // relative to rPosWait

GVL_XTS.StationParameter[nStationParameter].rReleaseDistance      :=     30.0; // relative to Mover.ActPos
GVL_XTS.StationParameter[nStationParameter].rGap                  :=     76.0;

//-----------------------------------------------------------------------------------------------------------------------------------------
nStationParameter := 23;
GVL_XTS.StationParameter[nStationParameter].sText                 := sStationText;
GVL_XTS.StationParameter[nStationParameter].rPosWait              :=   3582.0;  // absolute modulo position

GVL_XTS.StationParameter[nStationParameter].nConfiguredStopCount  :=      1;   // how many stops the mover has to make in this station
GVL_XTS.StationParameter[nStationParameter].rPosStop[1]           :=    760.0 + 161.0; // relative to rPosWait

GVL_XTS.StationParameter[nStationParameter].rReleaseDistance      :=     20.0; // relative to Mover.ActPos
GVL_XTS.StationParameter[nStationParameter].rGap                  :=     76.0;

//-----------------------------------------------------------------------------------------------------------------------------------------
nStationParameter := 24;
GVL_XTS.StationParameter[nStationParameter].sText                 := sStationText;
GVL_XTS.StationParameter[nStationParameter].rPosWait              :=   3582.0;  // absolute modulo position

GVL_XTS.StationParameter[nStationParameter].nConfiguredStopCount  :=      1;   // how many stops the mover has to make in this station
GVL_XTS.StationParameter[nStationParameter].rPosStop[1]           :=    836.0 + 161.0; // relative to rPosWait

GVL_XTS.StationParameter[nStationParameter].rReleaseDistance      :=     10.0; // relative to Mover.ActPos
GVL_XTS.StationParameter[nStationParameter].rGap                  :=     76.0;

GVL_XTS.StationParameter[nStationParameter].rVelo                 :=   1500.0;

//-----------------------------------------------------------------------------------------------------------------------------------------
//-----------------------------------------------------------------------------------------------------------------------------------------
//  BUFFER_OUTFEED_ROBOT
    sStationText  := TO_STRING(E_INSTANCE.BUFFER_OUTFEED);//'BUFFER_OUTFEED_ROBOT';
//-----------------------------------------------------------------------------------------------------------------------------------------
nStationParameter := 25;
GVL_XTS.StationParameter[nStationParameter].sText                 := sStationText;
GVL_XTS.StationParameter[nStationParameter].rPosWait              :=   3000.0;  // absolute modulo position

GVL_XTS.StationParameter[nStationParameter].nConfiguredStopCount  :=      1;   // how many stops the mover has to make in this station
GVL_XTS.StationParameter[nStationParameter].rPosStop[1]           :=      0.0; // relative to rPosWait

GVL_XTS.StationParameter[nStationParameter].rReleaseDistance      :=     -5.0; // relative to Mover.ActPos
GVL_XTS.StationParameter[nStationParameter].rGap                  :=     76.0;

//-----------------------------------------------------------------------------------------------------------------------------------------
//-----------------------------------------------------------------------------------------------------------------------------------------
//  OUTFEED_ROBOT_R1
    sStationText  := TO_STRING(E_INSTANCE.OUTFEED_ROBOT_R1);//'OUTFEED_ROBOT_R1';
//-----------------------------------------------------------------------------------------------------------------------------------------
nStationParameter := 26;
GVL_XTS.StationParameter[nStationParameter].sText                 := sStationText;
GVL_XTS.StationParameter[nStationParameter].rPosWait              :=   7000.0;  // absolute modulo position

GVL_XTS.StationParameter[nStationParameter].nConfiguredStopCount  :=      1;   // how many stops the mover has to make in this station
GVL_XTS.StationParameter[nStationParameter].rPosStop[1]           :=      0.0 + 160.0; // relative to rPosWait

GVL_XTS.StationParameter[nStationParameter].rReleaseDistance      :=    240.0; // relative to Mover.ActPos
GVL_XTS.StationParameter[nStationParameter].rGap                  :=     76.0;

//-----------------------------------------------------------------------------------------------------------------------------------------
nStationParameter := 27;
GVL_XTS.StationParameter[nStationParameter].sText                 := sStationText;
GVL_XTS.StationParameter[nStationParameter].rPosWait              :=   7000.0;  // absolute modulo position

GVL_XTS.StationParameter[nStationParameter].nConfiguredStopCount  :=      1;   // how many stops the mover has to make in this station
GVL_XTS.StationParameter[nStationParameter].rPosStop[1]           :=     80.0 + 160.0; // relative to rPosWait

GVL_XTS.StationParameter[nStationParameter].rReleaseDistance      :=    230.0; // relative to Mover.ActPos
GVL_XTS.StationParameter[nStationParameter].rGap                  :=     76.0;

//-----------------------------------------------------------------------------------------------------------------------------------------
nStationParameter := 28;
GVL_XTS.StationParameter[nStationParameter].sText                 := sStationText;
GVL_XTS.StationParameter[nStationParameter].rPosWait              :=   7000.0;  // absolute modulo position

GVL_XTS.StationParameter[nStationParameter].nConfiguredStopCount  :=      1;   // how many stops the mover has to make in this station
GVL_XTS.StationParameter[nStationParameter].rPosStop[1]           :=    160.0 + 160.0; // relative to rPosWait

GVL_XTS.StationParameter[nStationParameter].rReleaseDistance      :=    220.0; // relative to Mover.ActPos
GVL_XTS.StationParameter[nStationParameter].rGap                  :=     76.0;

//-----------------------------------------------------------------------------------------------------------------------------------------
nStationParameter := 29;
GVL_XTS.StationParameter[nStationParameter].sText                 := sStationText;
GVL_XTS.StationParameter[nStationParameter].rPosWait              :=   7000.0;  // absolute modulo position

GVL_XTS.StationParameter[nStationParameter].nConfiguredStopCount  :=      1;   // how many stops the mover has to make in this station
GVL_XTS.StationParameter[nStationParameter].rPosStop[1]           :=    240.0 + 160.0; // relative to rPosWait

GVL_XTS.StationParameter[nStationParameter].rReleaseDistance      :=    210.0; // relative to Mover.ActPos
GVL_XTS.StationParameter[nStationParameter].rGap                  :=     76.0;

//-----------------------------------------------------------------------------------------------------------------------------------------
nStationParameter := 30;
GVL_XTS.StationParameter[nStationParameter].sText                 := sStationText;
GVL_XTS.StationParameter[nStationParameter].rPosWait              :=   7000.0;  // absolute modulo position

GVL_XTS.StationParameter[nStationParameter].nConfiguredStopCount  :=      1;   // how many stops the mover has to make in this station
GVL_XTS.StationParameter[nStationParameter].rPosStop[1]           :=    320.0 + 160.0; // relative to rPosWait

GVL_XTS.StationParameter[nStationParameter].rReleaseDistance      :=    200.0; // relative to Mover.ActPos
GVL_XTS.StationParameter[nStationParameter].rGap                  :=     76.0;

//-----------------------------------------------------------------------------------------------------------------------------------------
nStationParameter := 31;
GVL_XTS.StationParameter[nStationParameter].sText                 := sStationText;
GVL_XTS.StationParameter[nStationParameter].rPosWait              :=   7000.0;  // absolute modulo position

GVL_XTS.StationParameter[nStationParameter].nConfiguredStopCount  :=      1;   // how many stops the mover has to make in this station
GVL_XTS.StationParameter[nStationParameter].rPosStop[1]           :=    400.0 + 160.0; // relative to rPosWait

GVL_XTS.StationParameter[nStationParameter].rReleaseDistance      :=    190.0; // relative to Mover.ActPos
GVL_XTS.StationParameter[nStationParameter].rGap                  :=     76.0;

//-----------------------------------------------------------------------------------------------------------------------------------------
nStationParameter := 32;
GVL_XTS.StationParameter[nStationParameter].sText                 := sStationText;
GVL_XTS.StationParameter[nStationParameter].rPosWait              :=   7000.0;  // absolute modulo position

GVL_XTS.StationParameter[nStationParameter].nConfiguredStopCount  :=      1;   // how many stops the mover has to make in this station
GVL_XTS.StationParameter[nStationParameter].rPosStop[1]           :=    480.0 + 160.0; // relative to rPosWait

GVL_XTS.StationParameter[nStationParameter].rReleaseDistance      :=    180.0; // relative to Mover.ActPos
GVL_XTS.StationParameter[nStationParameter].rGap                  :=     76.0;

//-----------------------------------------------------------------------------------------------------------------------------------------
nStationParameter := 33;
GVL_XTS.StationParameter[nStationParameter].sText                 := sStationText;
GVL_XTS.StationParameter[nStationParameter].rPosWait              :=   7000.0;  // absolute modulo position

GVL_XTS.StationParameter[nStationParameter].nConfiguredStopCount  :=      1;   // how many stops the mover has to make in this station
GVL_XTS.StationParameter[nStationParameter].rPosStop[1]           :=    560.0 + 160.0; // relative to rPosWait

GVL_XTS.StationParameter[nStationParameter].rReleaseDistance      :=    170.0; // relative to Mover.ActPos
GVL_XTS.StationParameter[nStationParameter].rGap                  :=     76.0;

//-----------------------------------------------------------------------------------------------------------------------------------------
nStationParameter := 34;
GVL_XTS.StationParameter[nStationParameter].sText                 := sStationText;
GVL_XTS.StationParameter[nStationParameter].rPosWait              :=   7000.0;  // absolute modulo position

GVL_XTS.StationParameter[nStationParameter].nConfiguredStopCount  :=      1;   // how many stops the mover has to make in this station
GVL_XTS.StationParameter[nStationParameter].rPosStop[1]           :=    640.0 + 160.0; // relative to rPosWait

GVL_XTS.StationParameter[nStationParameter].rReleaseDistance      :=    160.0; // relative to Mover.ActPos
GVL_XTS.StationParameter[nStationParameter].rGap                  :=     76.0;

//-----------------------------------------------------------------------------------------------------------------------------------------
nStationParameter := 35;
GVL_XTS.StationParameter[nStationParameter].sText                 := sStationText;
GVL_XTS.StationParameter[nStationParameter].rPosWait              :=   7000.0;  // absolute modulo position

GVL_XTS.StationParameter[nStationParameter].nConfiguredStopCount  :=      1;   // how many stops the mover has to make in this station
GVL_XTS.StationParameter[nStationParameter].rPosStop[1]           :=    720.0 + 160.0; // relative to rPosWait

GVL_XTS.StationParameter[nStationParameter].rReleaseDistance      :=    150.0; // relative to Mover.ActPos
GVL_XTS.StationParameter[nStationParameter].rGap                  :=     76.0;

//-----------------------------------------------------------------------------------------------------------------------------------------
nStationParameter := 36;
GVL_XTS.StationParameter[nStationParameter].sText                 := sStationText;
GVL_XTS.StationParameter[nStationParameter].rPosWait              :=   7000.0;  // absolute modulo position

GVL_XTS.StationParameter[nStationParameter].nConfiguredStopCount  :=      1;   // how many stops the mover has to make in this station
GVL_XTS.StationParameter[nStationParameter].rPosStop[1]           :=    800.0 + 160.0; // relative to rPosWait

GVL_XTS.StationParameter[nStationParameter].rReleaseDistance      :=    140.0; // relative to Mover.ActPos
GVL_XTS.StationParameter[nStationParameter].rGap                  :=     76.0;

//-----------------------------------------------------------------------------------------------------------------------------------------
nStationParameter := 37;
GVL_XTS.StationParameter[nStationParameter].sText                 := sStationText;
GVL_XTS.StationParameter[nStationParameter].rPosWait              :=   7000.0;  // absolute modulo position

GVL_XTS.StationParameter[nStationParameter].nConfiguredStopCount  :=      1;   // how many stops the mover has to make in this station
GVL_XTS.StationParameter[nStationParameter].rPosStop[1]           :=    880.0 + 160.0; // relative to rPosWait

GVL_XTS.StationParameter[nStationParameter].rReleaseDistance      :=    130.0; // relative to Mover.ActPos
GVL_XTS.StationParameter[nStationParameter].rGap                  :=     76.0;

//GVL_XTS.StationParameter[nStationParameter].rVelo                 :=   1500.0;

//-----------------------------------------------------------------------------------------------------------------------------------------
//-----------------------------------------------------------------------------------------------------------------------------------------
//  OUTFEED_ROBOT_R2
    sStationText  := TO_STRING(E_INSTANCE.OUTFEED_ROBOT_R2);//'OUTFEED_ROBOT_R2';
//-----------------------------------------------------------------------------------------------------------------------------------------
nStationParameter := 38;
GVL_XTS.StationParameter[nStationParameter].sText                 := sStationText;
GVL_XTS.StationParameter[nStationParameter].rPosWait              :=   7000.0;  // absolute modulo position

GVL_XTS.StationParameter[nStationParameter].nConfiguredStopCount  :=      1;   // how many stops the mover has to make in this station
GVL_XTS.StationParameter[nStationParameter].rPosStop[1]           :=      0.0 + 1120.0; // relative to rPosWait

GVL_XTS.StationParameter[nStationParameter].rReleaseDistance      :=    120.0; // relative to Mover.ActPos
GVL_XTS.StationParameter[nStationParameter].rGap                  :=     76.0;

//-----------------------------------------------------------------------------------------------------------------------------------------
nStationParameter := 39;
GVL_XTS.StationParameter[nStationParameter].sText                 := sStationText;
GVL_XTS.StationParameter[nStationParameter].rPosWait              :=   7000.0;  // absolute modulo position

GVL_XTS.StationParameter[nStationParameter].nConfiguredStopCount  :=      1;   // how many stops the mover has to make in this station
GVL_XTS.StationParameter[nStationParameter].rPosStop[1]           :=     80.0 + 1120.0; // relative to rPosWait

GVL_XTS.StationParameter[nStationParameter].rReleaseDistance      :=    110.0; // relative to Mover.ActPos
GVL_XTS.StationParameter[nStationParameter].rGap                  :=     76.0;

//-----------------------------------------------------------------------------------------------------------------------------------------
nStationParameter := 40;
GVL_XTS.StationParameter[nStationParameter].sText                 := sStationText;
GVL_XTS.StationParameter[nStationParameter].rPosWait              :=   7000.0;  // absolute modulo position

GVL_XTS.StationParameter[nStationParameter].nConfiguredStopCount  :=      1;   // how many stops the mover has to make in this station
GVL_XTS.StationParameter[nStationParameter].rPosStop[1]           :=    160.0 + 1120.0; // relative to rPosWait

GVL_XTS.StationParameter[nStationParameter].rReleaseDistance      :=    100.0; // relative to Mover.ActPos
GVL_XTS.StationParameter[nStationParameter].rGap                  :=     76.0;

//-----------------------------------------------------------------------------------------------------------------------------------------
nStationParameter := 41;
GVL_XTS.StationParameter[nStationParameter].sText                 := sStationText;
GVL_XTS.StationParameter[nStationParameter].rPosWait              :=   7000.0;  // absolute modulo position

GVL_XTS.StationParameter[nStationParameter].nConfiguredStopCount  :=      1;   // how many stops the mover has to make in this station
GVL_XTS.StationParameter[nStationParameter].rPosStop[1]           :=    240.0 + 1120.0; // relative to rPosWait

GVL_XTS.StationParameter[nStationParameter].rReleaseDistance      :=     90.0; // relative to Mover.ActPos
GVL_XTS.StationParameter[nStationParameter].rGap                  :=     76.0;

//-----------------------------------------------------------------------------------------------------------------------------------------
nStationParameter := 42;
GVL_XTS.StationParameter[nStationParameter].sText                 := sStationText;
GVL_XTS.StationParameter[nStationParameter].rPosWait              :=   7000.0;  // absolute modulo position

GVL_XTS.StationParameter[nStationParameter].nConfiguredStopCount  :=      1;   // how many stops the mover has to make in this station
GVL_XTS.StationParameter[nStationParameter].rPosStop[1]           :=    320.0 + 1120.0; // relative to rPosWait

GVL_XTS.StationParameter[nStationParameter].rReleaseDistance      :=     80.0; // relative to Mover.ActPos
GVL_XTS.StationParameter[nStationParameter].rGap                  :=     76.0;

//-----------------------------------------------------------------------------------------------------------------------------------------
nStationParameter := 43;
GVL_XTS.StationParameter[nStationParameter].sText                 := sStationText;
GVL_XTS.StationParameter[nStationParameter].rPosWait              :=   7000.0;  // absolute modulo position

GVL_XTS.StationParameter[nStationParameter].nConfiguredStopCount  :=      1;   // how many stops the mover has to make in this station
GVL_XTS.StationParameter[nStationParameter].rPosStop[1]           :=    400.0 + 1120.0; // relative to rPosWait

GVL_XTS.StationParameter[nStationParameter].rReleaseDistance      :=     70.0; // relative to Mover.ActPos
GVL_XTS.StationParameter[nStationParameter].rGap                  :=     76.0;

//-----------------------------------------------------------------------------------------------------------------------------------------
nStationParameter := 44;
GVL_XTS.StationParameter[nStationParameter].sText                 := sStationText;
GVL_XTS.StationParameter[nStationParameter].rPosWait              :=   7000.0;  // absolute modulo position

GVL_XTS.StationParameter[nStationParameter].nConfiguredStopCount  :=      1;   // how many stops the mover has to make in this station
GVL_XTS.StationParameter[nStationParameter].rPosStop[1]           :=    480.0 + 1120.0; // relative to rPosWait

GVL_XTS.StationParameter[nStationParameter].rReleaseDistance      :=     60.0; // relative to Mover.ActPos
GVL_XTS.StationParameter[nStationParameter].rGap                  :=     76.0;

//-----------------------------------------------------------------------------------------------------------------------------------------
nStationParameter := 45;
GVL_XTS.StationParameter[nStationParameter].sText                 := sStationText;
GVL_XTS.StationParameter[nStationParameter].rPosWait              :=   7000.0;  // absolute modulo position

GVL_XTS.StationParameter[nStationParameter].nConfiguredStopCount  :=      1;   // how many stops the mover has to make in this station
GVL_XTS.StationParameter[nStationParameter].rPosStop[1]           :=    560.0 + 1120.0; // relative to rPosWait

GVL_XTS.StationParameter[nStationParameter].rReleaseDistance      :=     50.0; // relative to Mover.ActPos
GVL_XTS.StationParameter[nStationParameter].rGap                  :=     76.0;

//-----------------------------------------------------------------------------------------------------------------------------------------
nStationParameter := 46;
GVL_XTS.StationParameter[nStationParameter].sText                 := sStationText;
GVL_XTS.StationParameter[nStationParameter].rPosWait              :=   7000.0;  // absolute modulo position

GVL_XTS.StationParameter[nStationParameter].nConfiguredStopCount  :=      1;   // how many stops the mover has to make in this station
GVL_XTS.StationParameter[nStationParameter].rPosStop[1]           :=    640.0 + 1120.0; // relative to rPosWait

GVL_XTS.StationParameter[nStationParameter].rReleaseDistance      :=     40.0; // relative to Mover.ActPos
GVL_XTS.StationParameter[nStationParameter].rGap                  :=     76.0;

//-----------------------------------------------------------------------------------------------------------------------------------------
nStationParameter := 47;
GVL_XTS.StationParameter[nStationParameter].sText                 := sStationText;
GVL_XTS.StationParameter[nStationParameter].rPosWait              :=   7000.0;  // absolute modulo position

GVL_XTS.StationParameter[nStationParameter].nConfiguredStopCount  :=      1;   // how many stops the mover has to make in this station
GVL_XTS.StationParameter[nStationParameter].rPosStop[1]           :=    720.0 + 1120.0; // relative to rPosWait

GVL_XTS.StationParameter[nStationParameter].rReleaseDistance      :=     30.0; // relative to Mover.ActPos
GVL_XTS.StationParameter[nStationParameter].rGap                  :=     76.0;

//-----------------------------------------------------------------------------------------------------------------------------------------
nStationParameter := 48;
GVL_XTS.StationParameter[nStationParameter].sText                 := sStationText;
GVL_XTS.StationParameter[nStationParameter].rPosWait              :=   7000.0;  // absolute modulo position

GVL_XTS.StationParameter[nStationParameter].nConfiguredStopCount  :=      1;   // how many stops the mover has to make in this station
GVL_XTS.StationParameter[nStationParameter].rPosStop[1]           :=    800.0 + 1120.0; // relative to rPosWait

GVL_XTS.StationParameter[nStationParameter].rReleaseDistance      :=     20.0; // relative to Mover.ActPos
GVL_XTS.StationParameter[nStationParameter].rGap                  :=     76.0;

//-----------------------------------------------------------------------------------------------------------------------------------------
nStationParameter := 49;
GVL_XTS.StationParameter[nStationParameter].sText                 := sStationText;
GVL_XTS.StationParameter[nStationParameter].rPosWait              :=   7000.0;  // absolute modulo position

GVL_XTS.StationParameter[nStationParameter].nConfiguredStopCount  :=      1;   // how many stops the mover has to make in this station
GVL_XTS.StationParameter[nStationParameter].rPosStop[1]           :=    880.0 + 1120.0; // relative to rPosWait

GVL_XTS.StationParameter[nStationParameter].rReleaseDistance      :=     10.0; // relative to Mover.ActPos
GVL_XTS.StationParameter[nStationParameter].rGap                  :=     76.0;

GVL_XTS.StationParameter[nStationParameter].rVelo                 :=   1500.0;


//-----------------------------------------------------------------------------------------------------------------------------------------
//-----------------------------------------------------------------------------------------------------------------------------------------
//  SENDER_SLOW is notin use in this example
    sStationText  := 'NOT_IN_USE';
//-----------------------------------------------------------------------------------------------------------------------------------------
//nStationParameter := 50;
//GVL_XTS.StationParameter[nStationParameter].sText                 := sStationText;
//GVL_XTS.StationParameter[nStationParameter].rPosWait              :=  10000.0;  // absolute modulo position

//GVL_XTS.StationParameter[nStationParameter].nConfiguredStopCount  :=      1;   // how many stops the mover has to make in this station
//GVL_XTS.StationParameter[nStationParameter].rPosStop[1]           :=      0.0; // relative to rPosWait

//GVL_XTS.StationParameter[nStationParameter].rReleaseDistance      :=     10.0; // relative to Mover.ActPos

//GVL_XTS.StationParameter[nStationParameter].rGap                  :=     76.0;
//GVL_XTS.StationParameter[nStationParameter].rVelo                 :=   1500.0;
//GVL_XTS.StationParameter[nStationParameter].rAccDec               :=  30000.0;
//GVL_XTS.StationParameter[nStationParameter].rJerk                 := 200000.0;

//-----------------------------------------------------------------------------------------------------------------------------------------
//-----------------------------------------------------------------------------------------------------------------------------------------
// SENDER_FAST
    sStationText  := TO_STRING(E_INSTANCE.SENDER_FAST);//'SENDER_FAST';
//-----------------------------------------------------------------------------------------------------------------------------------------
nStationParameter := 51;
GVL_XTS.StationParameter[nStationParameter].sText                 := sStationText;
GVL_XTS.StationParameter[nStationParameter].rPosWait              :=  12000.0;  // absolute modulo position

GVL_XTS.StationParameter[nStationParameter].nConfiguredStopCount  :=      1;   // how many stops the mover has to make in this station
GVL_XTS.StationParameter[nStationParameter].rPosStop[1]           :=      0.0; // relative to rPosWait

GVL_XTS.StationParameter[nStationParameter].rReleaseDistance      :=    -10.0; // relative to Mover.ActPos
GVL_XTS.StationParameter[nStationParameter].rGap                  :=     76.0;



//-----------------------------------------------------------------------------------------------------------------------------------------
//-----------------------------------------------------------------------------------------------------------------------------------------
//  SENDER_BUFFER_INFEED
    sStationText  := TO_STRING(E_INSTANCE.SENDER_BUFFER_INFEED);//'SENDER_BUFFER_INFEED';
//-----------------------------------------------------------------------------------------------------------------------------------------
nStationParameter := 52;
GVL_XTS.StationParameter[nStationParameter].sText                 := sStationText;
GVL_XTS.StationParameter[nStationParameter].rPosWait              :=  20500.0;  // absolute modulo position

GVL_XTS.StationParameter[nStationParameter].nConfiguredStopCount  :=      1;   // how many stops the mover has to make in this station
GVL_XTS.StationParameter[nStationParameter].rPosStop[1]           :=      0.0; // relative to rPosWait

GVL_XTS.StationParameter[nStationParameter].rReleaseDistance      :=    -10.0; // relative to Mover.ActPos
GVL_XTS.StationParameter[nStationParameter].rGap                  :=     76.0;

GVL_XTS.StationParameter[nStationParameter].rVelo                 :=   1500.0;
GVL_XTS.StationParameter[nStationParameter].rAccDec               :=  15000.0;


//-----------------------------------------------------------------------------------------------------------------------------------------
//-----------------------------------------------------------------------------------------------------------------------------------------
//  BUFFER_INFEED
    sStationText  := TO_STRING(E_INSTANCE.BUFFER_INFEED);//'BUFFER_INFEED';
//-----------------------------------------------------------------------------------------------------------------------------------------
nStationParameter := 53;
GVL_XTS.StationParameter[nStationParameter].sText                 := sStationText;
GVL_XTS.StationParameter[nStationParameter].rPosWait              :=    1200.0;  // absolute modulo position

GVL_XTS.StationParameter[nStationParameter].nConfiguredStopCount  :=      1;   // how many stops the mover has to make in this station
GVL_XTS.StationParameter[nStationParameter].rPosStop[1]           :=      0.0; // relative to rPosWait

GVL_XTS.StationParameter[nStationParameter].rReleaseDistance      :=    -10.0; // relative to Mover.ActPos
GVL_XTS.StationParameter[nStationParameter].rGap                  :=    76.0;

GVL_XTS.StationParameter[nStationParameter].rVelo                 :=   1250.0;
END_ACTION

ACTION J_100000_V3500:
//-----------------------------------------------------------------------------
//
//  HAUD 2024.06.12
//
// 
//  - hard coded station parameter
//-----------------------------------------------------------------------------
//-----------------------------------------------------------------------------

FOR nStationParameter := 1 TO MAX_STATION
DO
  GVL_XTS.StationParameter[nStationParameter].rVelo               :=   3500.0;
  GVL_XTS.StationParameter[nStationParameter].rAccDec             :=  rAcc;
  GVL_XTS.StationParameter[nStationParameter].rJerk               := 100000.0;
END_FOR 

//-----------------------------------------------------------------------------------------------------------------------------------------
//  INFEED
    sStationText  := TO_STRING(E_INSTANCE.INFEED);//'INFEED';
//-----------------------------------------------------------------------------------------------------------------------------------------
nStationParameter := 1;
GVL_XTS.StationParameter[nStationParameter].sText                 := sStationText;
GVL_XTS.StationParameter[nStationParameter].rPosWait              :=    1250.0;  // absolute modulo position

GVL_XTS.StationParameter[nStationParameter].nConfiguredStopCount  :=      1;   // how many stops the mover has to make in this station
GVL_XTS.StationParameter[nStationParameter].rPosStop[1]           :=      0.0 + 176.0; // relative to rPosWait

GVL_XTS.StationParameter[nStationParameter].rReleaseDistance      :=    300.0; // relative to Mover.ActPos
GVL_XTS.StationParameter[nStationParameter].rGap                  :=     76.0;

//-----------------------------------------------------------------------------------------------------------------------------------------
nStationParameter := 2;
GVL_XTS.StationParameter[nStationParameter].sText                 := sStationText;
GVL_XTS.StationParameter[nStationParameter].rPosWait              :=    1250.0; // absolute modulo position

GVL_XTS.StationParameter[nStationParameter].nConfiguredStopCount  :=      1;   // how many stops the mover has to make in this station
GVL_XTS.StationParameter[nStationParameter].rPosStop[1]           :=     76.0 + 176.0; // relative to rPosWait

GVL_XTS.StationParameter[nStationParameter].rReleaseDistance      :=    275.0; // relative to Mover.ActPos
GVL_XTS.StationParameter[nStationParameter].rGap                  :=     76.0;

//-----------------------------------------------------------------------------------------------------------------------------------------
nStationParameter := 3;
GVL_XTS.StationParameter[nStationParameter].sText                 := sStationText;
GVL_XTS.StationParameter[nStationParameter].rPosWait              :=    1250.0; // absolute modulo position

GVL_XTS.StationParameter[nStationParameter].nConfiguredStopCount  :=      1;   // how many stops the mover has to make in this station
GVL_XTS.StationParameter[nStationParameter].rPosStop[1]           :=    152.0 + 176.0; // relative to rPosWait

GVL_XTS.StationParameter[nStationParameter].rReleaseDistance      :=    250.0; // relative to Mover.ActPos
GVL_XTS.StationParameter[nStationParameter].rGap                  :=     76.0;

//-----------------------------------------------------------------------------------------------------------------------------------------
nStationParameter := 4;
GVL_XTS.StationParameter[nStationParameter].sText                 := sStationText;
GVL_XTS.StationParameter[nStationParameter].rPosWait              :=   1250.0;  // absolute modulo position

GVL_XTS.StationParameter[nStationParameter].nConfiguredStopCount  :=      1;   // how many stops the mover has to make in this station
GVL_XTS.StationParameter[nStationParameter].rPosStop[1]           :=    228.0 + 176.0; // relative to rPosWait

GVL_XTS.StationParameter[nStationParameter].rReleaseDistance      :=    225.0; // relative to Mover.ActPos
GVL_XTS.StationParameter[nStationParameter].rGap                  :=     76.0;

//-----------------------------------------------------------------------------------------------------------------------------------------
nStationParameter := 5;
GVL_XTS.StationParameter[nStationParameter].sText                 := sStationText;
GVL_XTS.StationParameter[nStationParameter].rPosWait              :=   1250.0;  // absolute modulo position

GVL_XTS.StationParameter[nStationParameter].nConfiguredStopCount  :=      1;   // how many stops the mover has to make in this station
GVL_XTS.StationParameter[nStationParameter].rPosStop[1]           :=    304.0 + 176.0; // relative to rPosWait

GVL_XTS.StationParameter[nStationParameter].rReleaseDistance      :=    200.0; // relative to Mover.ActPos
GVL_XTS.StationParameter[nStationParameter].rGap                  :=     76.0;

//-----------------------------------------------------------------------------------------------------------------------------------------
nStationParameter := 6;
GVL_XTS.StationParameter[nStationParameter].sText                 := sStationText;
GVL_XTS.StationParameter[nStationParameter].rPosWait              :=   1250.0;  // absolute modulo position

GVL_XTS.StationParameter[nStationParameter].nConfiguredStopCount  :=      1;   // how many stops the mover has to make in this station
GVL_XTS.StationParameter[nStationParameter].rPosStop[1]           :=    380.0 + 176.0; // relative to rPosWait

GVL_XTS.StationParameter[nStationParameter].rReleaseDistance      :=    175.0; // relative to Mover.ActPos
GVL_XTS.StationParameter[nStationParameter].rGap                  :=     76.0;

//-----------------------------------------------------------------------------------------------------------------------------------------
nStationParameter := 7;
GVL_XTS.StationParameter[nStationParameter].sText                 := sStationText;
GVL_XTS.StationParameter[nStationParameter].rPosWait              :=   1250.0;  // absolute modulo position

GVL_XTS.StationParameter[nStationParameter].nConfiguredStopCount  :=      1;   // how many stops the mover has to make in this station
GVL_XTS.StationParameter[nStationParameter].rPosStop[1]           :=    456.0 + 176.0; // relative to rPosWait

GVL_XTS.StationParameter[nStationParameter].rReleaseDistance      :=    150.0; // relative to Mover.ActPos
GVL_XTS.StationParameter[nStationParameter].rGap                  :=     76.0;

//-----------------------------------------------------------------------------------------------------------------------------------------
nStationParameter := 8;
GVL_XTS.StationParameter[nStationParameter].sText                 := sStationText;
GVL_XTS.StationParameter[nStationParameter].rPosWait              :=   1250.0;  // absolute modulo position

GVL_XTS.StationParameter[nStationParameter].nConfiguredStopCount  :=      1;   // how many stops the mover has to make in this station
GVL_XTS.StationParameter[nStationParameter].rPosStop[1]           :=    532.0 + 176.0; // relative to rPosWait

GVL_XTS.StationParameter[nStationParameter].rReleaseDistance      :=    125.0; // relative to Mover.ActPos
GVL_XTS.StationParameter[nStationParameter].rGap                  :=     76.0;

//-----------------------------------------------------------------------------------------------------------------------------------------
nStationParameter := 9;
GVL_XTS.StationParameter[nStationParameter].sText                 := sStationText;
GVL_XTS.StationParameter[nStationParameter].rPosWait              :=   1250.0;  // absolute modulo position

GVL_XTS.StationParameter[nStationParameter].nConfiguredStopCount  :=      1;   // how many stops the mover has to make in this station
GVL_XTS.StationParameter[nStationParameter].rPosStop[1]           :=    608.0 + 176.0; // relative to rPosWait

GVL_XTS.StationParameter[nStationParameter].rReleaseDistance      :=    100.0; // relative to Mover.ActPos
GVL_XTS.StationParameter[nStationParameter].rGap                  :=     76.0;

//-----------------------------------------------------------------------------------------------------------------------------------------
nStationParameter := 10;
GVL_XTS.StationParameter[nStationParameter].sText                 := sStationText;
GVL_XTS.StationParameter[nStationParameter].rPosWait              :=   1250.0;  // absolute modulo position

GVL_XTS.StationParameter[nStationParameter].nConfiguredStopCount  :=      1;   // how many stops the mover has to make in this station
GVL_XTS.StationParameter[nStationParameter].rPosStop[1]           :=    684.0 + 176.0; // relative to rPosWait

GVL_XTS.StationParameter[nStationParameter].rReleaseDistance      :=     75.0; // relative to Mover.ActPos
GVL_XTS.StationParameter[nStationParameter].rGap                  :=     76.0;

//-----------------------------------------------------------------------------------------------------------------------------------------
nStationParameter := 11;
GVL_XTS.StationParameter[nStationParameter].sText                 := sStationText;
GVL_XTS.StationParameter[nStationParameter].rPosWait              :=   1250.0;  // absolute modulo position

GVL_XTS.StationParameter[nStationParameter].nConfiguredStopCount  :=      1;   // how many stops the mover has to make in this station
GVL_XTS.StationParameter[nStationParameter].rPosStop[1]           :=    760.0 + 176.0; // relative to rPosWait

GVL_XTS.StationParameter[nStationParameter].rReleaseDistance      :=     50.0; // relative to Mover.ActPos
GVL_XTS.StationParameter[nStationParameter].rGap                  :=     76.0;

//-----------------------------------------------------------------------------------------------------------------------------------------
nStationParameter := 12;
GVL_XTS.StationParameter[nStationParameter].sText                 := sStationText;
GVL_XTS.StationParameter[nStationParameter].rPosWait              :=   1250.0;  // absolute modulo position

GVL_XTS.StationParameter[nStationParameter].nConfiguredStopCount  :=      1;   // how many stops the mover has to make in this station
GVL_XTS.StationParameter[nStationParameter].rPosStop[1]           :=    836.0 + 176.0; // relative to rPosWait

GVL_XTS.StationParameter[nStationParameter].rReleaseDistance      :=     10.0; // relative to Mover.ActPos
GVL_XTS.StationParameter[nStationParameter].rGap                  :=     76.0;

//-----------------------------------------------------------------------------------------------------------------------------------------
//-----------------------------------------------------------------------------------------------------------------------------------------
//  OUTFEED_CLAMP (not in use in this example)
    sStationText  := 'OUTFEED_CLAMP';
//-----------------------------------------------------------------------------------------------------------------------------------------
nStationParameter := 13;
GVL_XTS.StationParameter[nStationParameter].sText                 := sStationText;
GVL_XTS.StationParameter[nStationParameter].rPosWait              :=   3582.0;  // absolute modulo position

GVL_XTS.StationParameter[nStationParameter].nConfiguredStopCount  :=      1;   // how many stops the mover has to make in this station
GVL_XTS.StationParameter[nStationParameter].rPosStop[1]           :=      0.0 + 161.0; // relative to rPosWait

GVL_XTS.StationParameter[nStationParameter].rReleaseDistance      :=    120.0; // relative to Mover.ActPos
GVL_XTS.StationParameter[nStationParameter].rGap                  :=     76.0;

//-----------------------------------------------------------------------------------------------------------------------------------------
nStationParameter := 14;
GVL_XTS.StationParameter[nStationParameter].sText                 := sStationText;
GVL_XTS.StationParameter[nStationParameter].rPosWait              :=   3582.0;  // absolute modulo position

GVL_XTS.StationParameter[nStationParameter].nConfiguredStopCount  :=      1;   // how many stops the mover has to make in this station
GVL_XTS.StationParameter[nStationParameter].rPosStop[1]           :=     76.0 + 161.0; // relative to rPosWait

GVL_XTS.StationParameter[nStationParameter].rReleaseDistance      :=    110.0; // relative to Mover.ActPos
GVL_XTS.StationParameter[nStationParameter].rGap                  :=     76.0;

//-----------------------------------------------------------------------------------------------------------------------------------------
nStationParameter := 15;
GVL_XTS.StationParameter[nStationParameter].sText                 := sStationText;
GVL_XTS.StationParameter[nStationParameter].rPosWait              :=   3582.0;  // absolute modulo position

GVL_XTS.StationParameter[nStationParameter].nConfiguredStopCount  :=      1;   // how many stops the mover has to make in this station
GVL_XTS.StationParameter[nStationParameter].rPosStop[1]           :=    152.0 + 161.0; // relative to rPosWait

GVL_XTS.StationParameter[nStationParameter].rReleaseDistance      :=    100.0; // relative to Mover.ActPos
GVL_XTS.StationParameter[nStationParameter].rGap                  :=     76.0;

//-----------------------------------------------------------------------------------------------------------------------------------------
nStationParameter := 16;
GVL_XTS.StationParameter[nStationParameter].sText                 := sStationText;
GVL_XTS.StationParameter[nStationParameter].rPosWait              :=   3582.0;  // absolute modulo position

